{attribute 'enable_dynamic_creation'}
FUNCTION_BLOCK EspHost IMPLEMENTS ITF_EspHost, ITF_Node
VAR
	
	// Node information
	LastNode					: ITF_Node;
	NextNode					: ITF_Node;
	PositionInList				: UINT;
	
	
	
	// ESP information
	ObjectId					: ULINT;
	PacketsReceivedCount		: ULINT;
	LastReceivedTimer			: TON;
	DistanceFromMaster			: BYTE;
	Data						: ARRAY [1..1000, 1..1000] OF BYTE;
	
END_VAR

{warning 'Add method implementation '}
METHOD CyclicUpdate : BOOL
LastReceivedTimer(PT := T#5S);
END_METHOD

METHOD GetLastNode : ITF_Node
GetLastNode := LastNode;

RETURN;
END_METHOD

METHOD GetMyPointer : PVOID
GetMyPointer := ADR(THIS^);
END_METHOD

METHOD GetNextNode : ITF_Node
GetNextNode := NextNode;

RETURN;
END_METHOD

METHOD GetPositionInList : UINT
GetPositionInList := PositionInList;

RETURN;
END_METHOD

METHOD HasTimedOut : BOOL
IF LastReceivedTimer.Q THEN
	
	HasTimedOut := TRUE;
	
ELSE
	
	HasTimedOut := FALSE;

END_IF
END_METHOD

{warning 'Add property implementation'}
PROPERTY PacketsReceived : ULINT
GET
PacketsReceived := THIS^.PacketsReceivedCount;
END_GET
SET
END_SET
END_PROPERTY

METHOD SetLastNode : BOOL
VAR_INPUT
	Node	: ITF_Node;
END_VAR
LastNode := Node;

SetLastNode := TRUE;

RETURN;
END_METHOD

METHOD SetNextNode : BOOL
VAR_INPUT
	Node	: ITF_Node;
END_VAR
NextNode := Node;

SetNextNode := TRUE;

RETURN;
END_METHOD

METHOD SetPositionInList : BOOL
VAR_INPUT
	Index	: UINT;
END_VAR
PositionInList := Index;

SetPositionInList := TRUE;

RETURN;
END_METHOD

{warning 'Add property implementation'}
PROPERTY Uid : ULINT
GET
Uid := THIS^.ObjectId;
END_GET
SET
IF THIS^.ObjectId = 0 THEN

	THIS^.ObjectId := Uid;	

END_IF
END_SET
END_PROPERTY

END_FUNCTION_BLOCK

(* stored: Version 1.1.0.1
   POU EspHost: Id {b3fe8272-bf4b-4466-9679-d62f1ddfa137}, SpecialFunc None
   Folder ITF_EspHost: Id {3e1ad894-296e-4a6b-bccd-5c988016ec11}
   Folder ITF_Node: Id {1137c9b1-75b7-4fc7-8824-f307a94e0aea}
   Method CyclicUpdate: Id {bd38af97-0931-41e0-88e6-255853f43dce}
   Method GetLastNode: Id {40659afe-16b7-4736-a59c-d79330896cb4}
   Method GetMyPointer: Id {278de2df-56c5-465c-bf04-1733d5508c6f}
   Method GetNextNode: Id {b8dfccf7-235a-47d0-aadc-c1a9701a3cc6}
   Method GetPositionInList: Id {30f4f578-233f-46f8-bc0a-f0861309c4dc}
   Method HasTimedOut: Id {603925a8-3f9a-4299-b307-beb68e1cd417}
   Property PacketsReceived: Id {1004878e-e09d-4d3a-a68d-5c1688ca98fe}
   Get Get: Id {1ebebfe9-85c0-4d64-8f07-1fc763760c90}
   Set Set: Id {1068f119-a0ad-4960-b007-c8dae36816f7}
   Method SetLastNode: Id {c5dd63a9-ada1-4b64-97ef-df115a746a4e}
   Method SetNextNode: Id {c54b15ba-0586-46b9-8a8b-5078fec904e4}
   Method SetPositionInList: Id {d2bd9100-91b9-4c94-b69e-66d983599699}
   Property Uid: Id {8c151426-fdc1-4292-aeff-50fb5feba438}
   Get Get: Id {10c3a14d-374b-43eb-826b-11fbe9d89326}
   Set Set: Id {faef1185-67a9-4f19-9e8f-404f70500a9d} *)
